(* Logix 5000 project; controller Receptivo vendor 1 type 14 code 106 rev 30.11; software revision 30.00; part 8 of 10 *)
(* tags used below, declared in another part *)
   Cantidad_de_Productos : DINT;
   codigo_capturado_1 : BOOL;
   codigo_capturado_2 : BOOL;
   codigo_capturado_3 : BOOL;
   codigo_capturado_4 : BOOL;
   Cont_Prod_1 : DINT;
   Cont_Prod_2 : DINT;
   Cont_Prod_3 : DINT;
   Cont_Prod_4 : DINT;
   Datos_1_Manual : BOOL;
   Datos_2_Manual : BOOL;
   Datos_3_Manual : BOOL;
   Datos_4_Manual : BOOL;
   EAN14_1 : Codigo_Barras;
   EAN14_2 : Codigo_Barras;
   EAN14_3 : Codigo_Barras;
   EAN14_4 : Codigo_Barras;
   Estacion_1_GCola_1 : UDT_COLA;
   Estacion_1_General : UDT_GENERAL;
   Estacion_2_GCola_1 : UDT_COLA;
   Estacion_2_General : UDT_GENERAL;
   Estacion_3_GCola_1 : UDT_COLA;
   Estacion_3_General : UDT_GENERAL;
   Estacion_4_GCola_1 : UDT_COLA;
   Estacion_4_General : UDT_GENERAL;
   No_existe : Descripcion;
   PB_Tare_Station_1 : BOOL;
   PB_Tare_Station_2 : BOOL;
   PESO_REAL_1 : DINT;
   PESO_REAL_2 : DINT;
   Producto1 : UDT_Inventario;
   Producto2 : UDT_Inventario;
   Producto3 : UDT_Inventario;
   Producto4 : UDT_Inventario;
   Producto_Codigo_Aceite_1 : DINT;
   Producto_Codigo_Aceite_2 : DINT;
   Producto_Codigo_Aceite_3 : DINT;
   Producto_Codigo_Aceite_4 : DINT;
   Productos : UDT_Maestro[300];
   QAD_1 : STRING;
   QAD_2 : STRING;
   QAD_3 : STRING;
   QAD_4 : STRING;
   Sin_Codigo : UDT_QAD;
   Station1_Tare_OK : BOOL;
   Station2_Tare_OK : BOOL;
   Tara_Fecha_Estacion_1 : Hora_y_Fecha;
   Tara_Fecha_Estacion_2 : Hora_y_Fecha;
   Tare_Station_1_Write : DINT;
   Tare_Station_2_Write : DINT;
   WPM1_Heartbeat : DINT;
   WPM1_Heartbeat_Error : BOOL;
   WPM1_Status : WPM_Status;
   WPM2_Heartbeat : DINT;
   WPM2_Heartbeat_Error : BOOL;
   WPM2_Status : WPM_Status;
   WPM_1_Selected : DINT;
   WPM_1_Status_Aux : DINT;
   WPM_2_COUNT_ANTERIOR : DINT;
   WPM_2_Selected : DINT;
   WPM_2_Status_Aux : DINT;
   Zero : DINT;

PROGRAM Manejo_Productos   (* main routine Inicial_Productos *)
VAR
   Final_captura_1 : BOOL;
   Final_captura_2 : BOOL;
   Final_captura_3 : BOOL;
   Final_captura_4 : BOOL;
   index_1 : DINT := 1;
   index_2 : DINT := 1;
   index_3 : DINT := 1;
   index_4 : DINT := 1;
   limite : BOOL := 1;
   ons_busca_1 : BOOL;
   ons_busca_2 : BOOL;
   ons_busca_3 : BOOL;
   ons_busca_4 : BOOL;
   ONS_CAPTURA : BOOL := 1;
   ONS_CAPTURA2 : BOOL;
   ONS_CAPTURA3 : BOOL;
   ONS_CAPTURA4 : BOOL;
   ons_captura_1 : BOOL;
   ons_dato_manual_1 : BOOL;
   ons_search : BOOL;
   vacio : STRING;
   victor : BOOL := 1;
END_VAR

ROUTINE Buscar_Productos_1   (* ladder *)
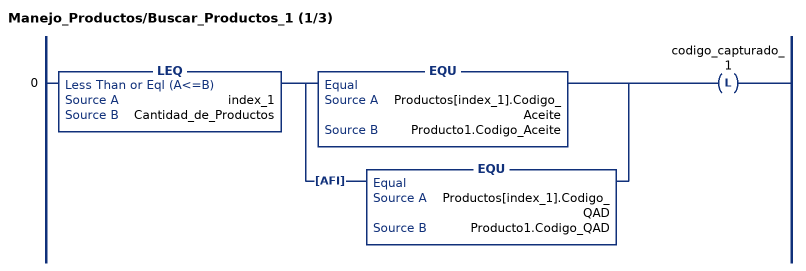
   0: LEQ(index_1,Cantidad_de_Productos)[EQU(Productos[index_1].Codigo_Aceite,Producto1.Codigo_Aceite) ,AFI() EQU(Productos[index_1].Codigo_QAD,Producto1.Codigo_QAD) ]OTL(codigo_capturado_1);
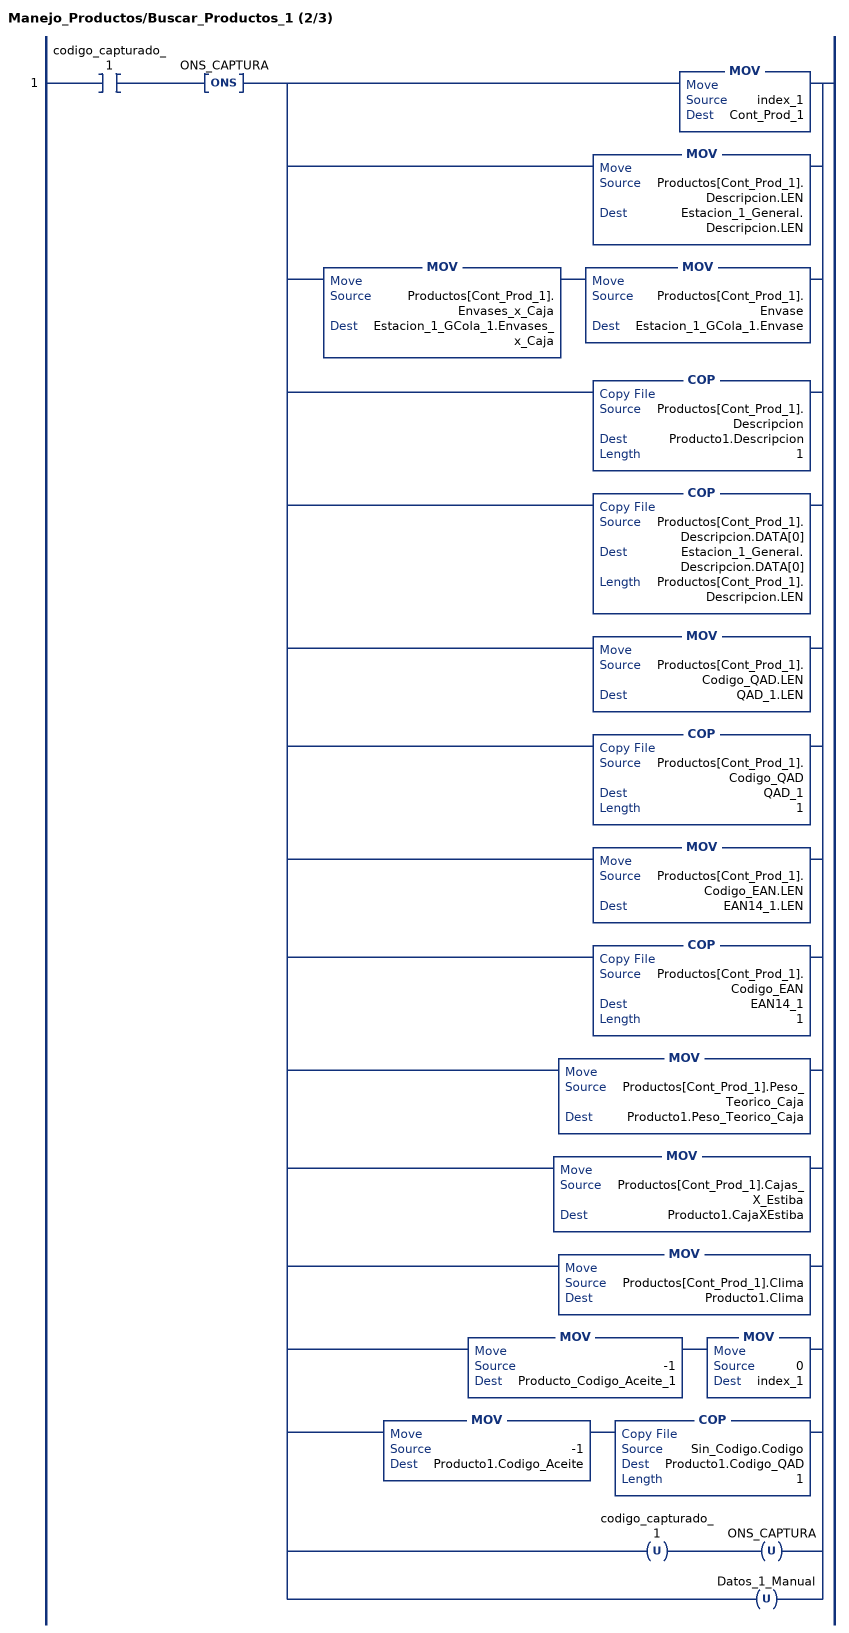
   1: XIC(codigo_capturado_1)ONS(ONS_CAPTURA)[MOV(index_1,Cont_Prod_1) ,MOV(Productos[Cont_Prod_1].Descripcion.LEN,Estacion_1_General.Descripcion.LEN) ,MOV(Productos[Cont_Prod_1].Envases_x_Caja,Estacion_1_GCola_1.Envases_x_Caja) MOV(Productos[Cont_Prod_1].Envase,Estacion_1_GCola_1.Envase) ,COP(Productos[Cont_Prod_1].Descripcion,Producto1.Descripcion,1) ,COP(Productos[Cont_Prod_1].Descripcion.DATA[0],Estacion_1_General.Descripcion.DATA[0],Productos[Cont_Prod_1].Descripcion.LEN) ,MOV(Productos[Cont_Prod_1].Codigo_QAD.LEN,QAD_1.LEN) ,COP(Productos[Cont_Prod_1].Codigo_QAD,QAD_1,1) ,MOV(Productos[Cont_Prod_1].Codigo_EAN.LEN,EAN14_1.LEN) ,COP(Productos[Cont_Prod_1].Codigo_EAN,EAN14_1,1) ,MOV(Productos[Cont_Prod_1].Peso_Teorico_Caja,Producto1.Peso_Teorico_Caja) ,MOV(Productos[Cont_Prod_1].Cajas_X_Estiba,Producto1.CajaXEstiba) ,MOV(Productos[Cont_Prod_1].Clima,Producto1.Clima) ,MOV(-1,Producto_Codigo_Aceite_1) MOV(0,index_1) ,MOV(-1,Producto1.Codigo_Aceite) COP(Sin_Codigo.Codigo,Producto1.Codigo_QAD,1) ,OTU(codigo_capturado_1) OTU(ONS_CAPTURA) ,OTU(Datos_1_Manual) ];
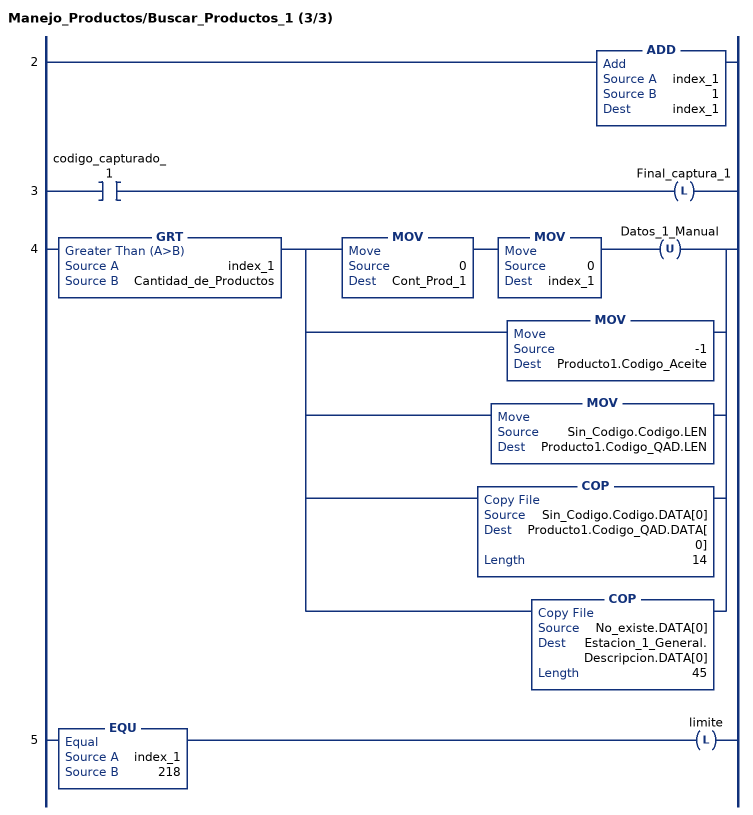
   2: ADD(index_1,1,index_1);
   3: XIC(codigo_capturado_1)OTL(Final_captura_1);
   4: GRT(index_1,Cantidad_de_Productos)[MOV(0,Cont_Prod_1) MOV(0,index_1) OTU(Datos_1_Manual) ,MOV(-1,Producto1.Codigo_Aceite) ,MOV(Sin_Codigo.Codigo.LEN,Producto1.Codigo_QAD.LEN) ,COP(Sin_Codigo.Codigo.DATA[0],Producto1.Codigo_QAD.DATA[0],14) ,COP(No_existe.DATA[0],Estacion_1_General.Descripcion.DATA[0],45) ];
   5: EQU(index_1,218)OTL(limite);
END_ROUTINE

ROUTINE Buscar_Productos_2   (* ladder *)
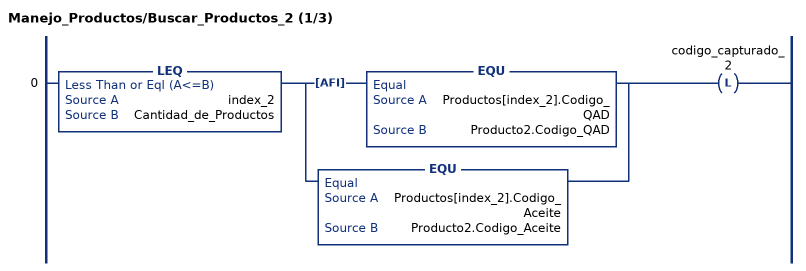
   0: LEQ(index_2,Cantidad_de_Productos)[AFI() EQU(Productos[index_2].Codigo_QAD,Producto2.Codigo_QAD) ,EQU(Productos[index_2].Codigo_Aceite,Producto2.Codigo_Aceite) ]OTL(codigo_capturado_2);
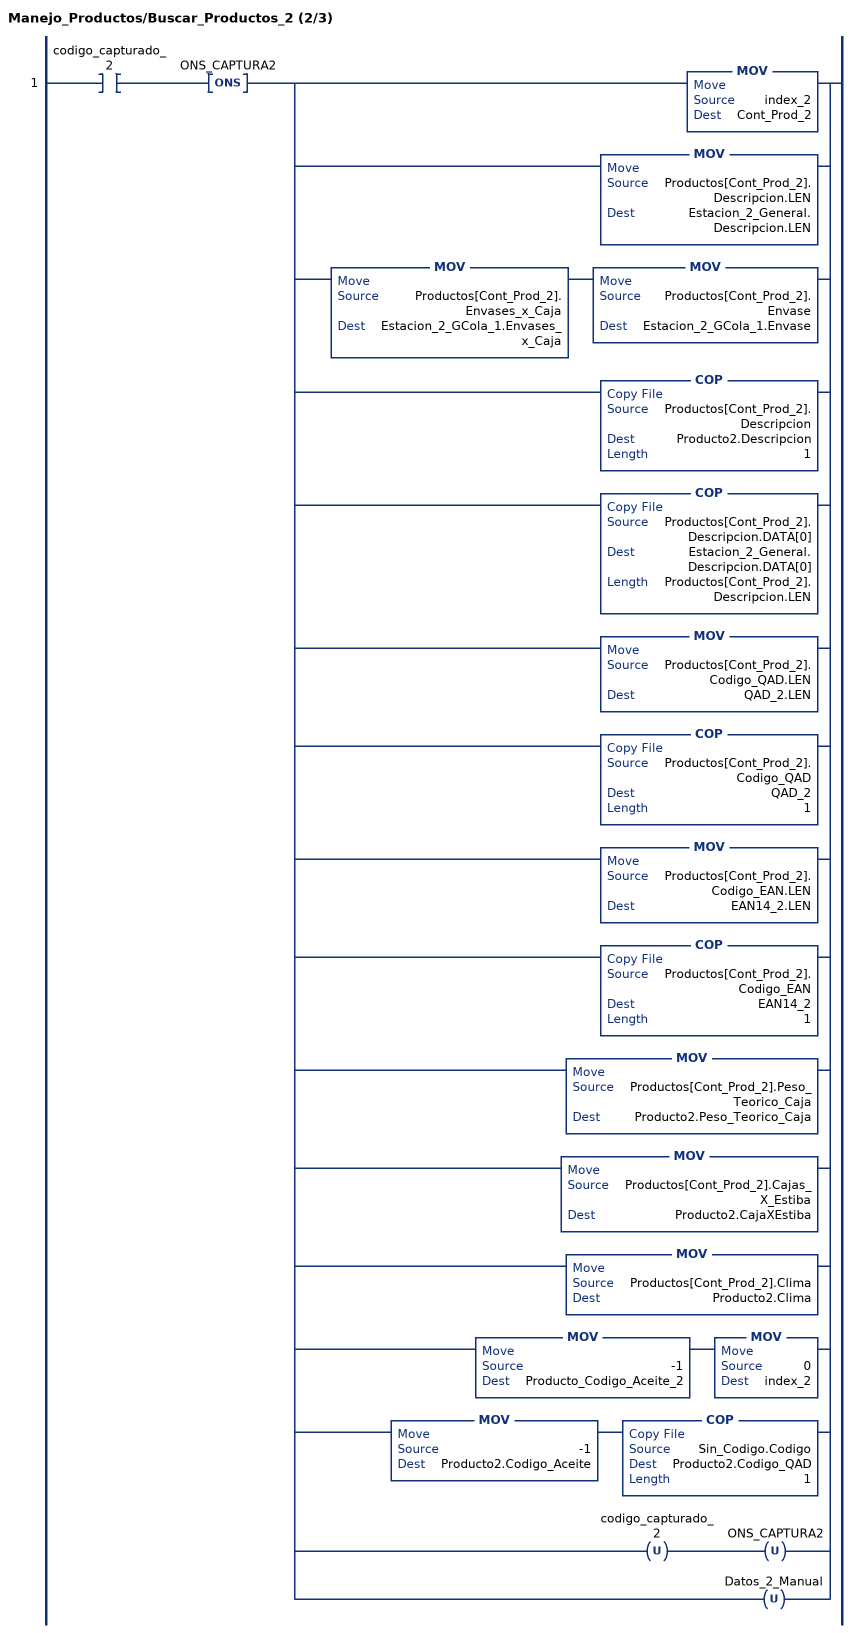
   1: XIC(codigo_capturado_2)ONS(ONS_CAPTURA2)[MOV(index_2,Cont_Prod_2) ,MOV(Productos[Cont_Prod_2].Descripcion.LEN,Estacion_2_General.Descripcion.LEN) ,MOV(Productos[Cont_Prod_2].Envases_x_Caja,Estacion_2_GCola_1.Envases_x_Caja) MOV(Productos[Cont_Prod_2].Envase,Estacion_2_GCola_1.Envase) ,COP(Productos[Cont_Prod_2].Descripcion,Producto2.Descripcion,1) ,COP(Productos[Cont_Prod_2].Descripcion.DATA[0],Estacion_2_General.Descripcion.DATA[0],Productos[Cont_Prod_2].Descripcion.LEN) ,MOV(Productos[Cont_Prod_2].Codigo_QAD.LEN,QAD_2.LEN) ,COP(Productos[Cont_Prod_2].Codigo_QAD,QAD_2,1) ,MOV(Productos[Cont_Prod_2].Codigo_EAN.LEN,EAN14_2.LEN) ,COP(Productos[Cont_Prod_2].Codigo_EAN,EAN14_2,1) ,MOV(Productos[Cont_Prod_2].Peso_Teorico_Caja,Producto2.Peso_Teorico_Caja) ,MOV(Productos[Cont_Prod_2].Cajas_X_Estiba,Producto2.CajaXEstiba) ,MOV(Productos[Cont_Prod_2].Clima,Producto2.Clima) ,MOV(-1,Producto_Codigo_Aceite_2) MOV(0,index_2) ,MOV(-1,Producto2.Codigo_Aceite) COP(Sin_Codigo.Codigo,Producto2.Codigo_QAD,1) ,OTU(codigo_capturado_2) OTU(ONS_CAPTURA2) ,OTU(Datos_2_Manual) ];
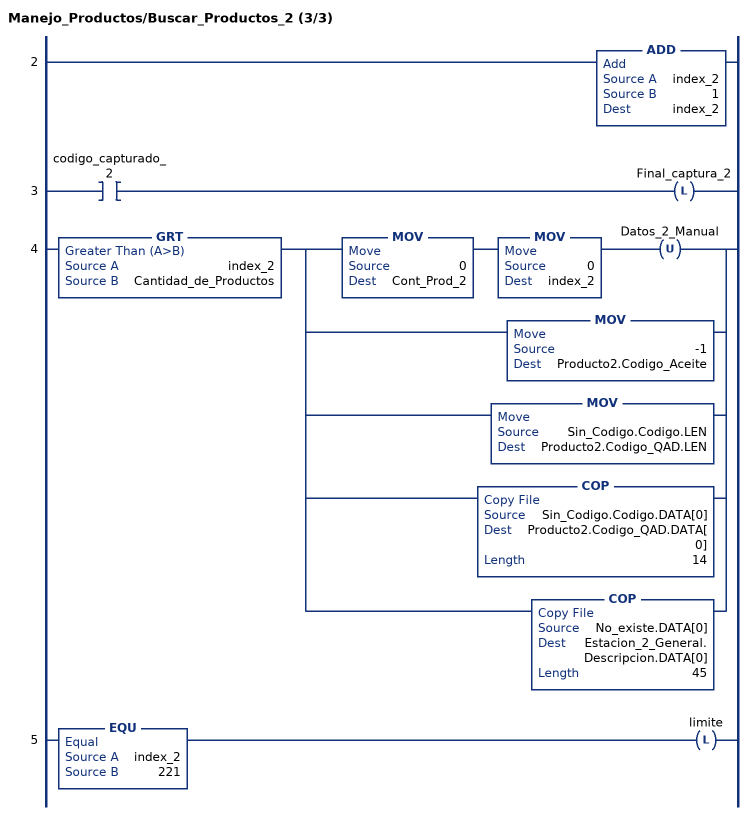
   2: ADD(index_2,1,index_2);
   3: XIC(codigo_capturado_2)OTL(Final_captura_2);
   4: GRT(index_2,Cantidad_de_Productos)[MOV(0,Cont_Prod_2) MOV(0,index_2) OTU(Datos_2_Manual) ,MOV(-1,Producto2.Codigo_Aceite) ,MOV(Sin_Codigo.Codigo.LEN,Producto2.Codigo_QAD.LEN) ,COP(Sin_Codigo.Codigo.DATA[0],Producto2.Codigo_QAD.DATA[0],14) ,COP(No_existe.DATA[0],Estacion_2_General.Descripcion.DATA[0],45) ];
   5: EQU(index_2,221)OTL(limite);
END_ROUTINE

ROUTINE Buscar_Productos_3   (* ladder *)
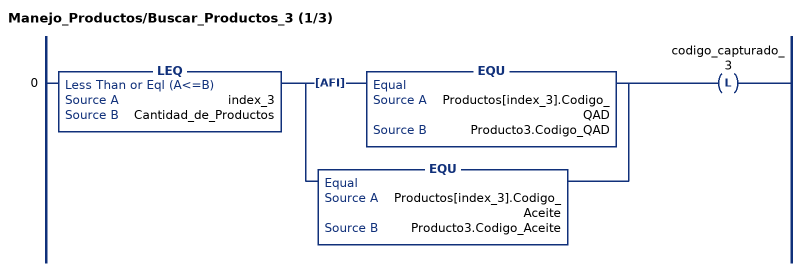
   0: LEQ(index_3,Cantidad_de_Productos)[AFI() EQU(Productos[index_3].Codigo_QAD,Producto3.Codigo_QAD) ,EQU(Productos[index_3].Codigo_Aceite,Producto3.Codigo_Aceite) ]OTL(codigo_capturado_3);
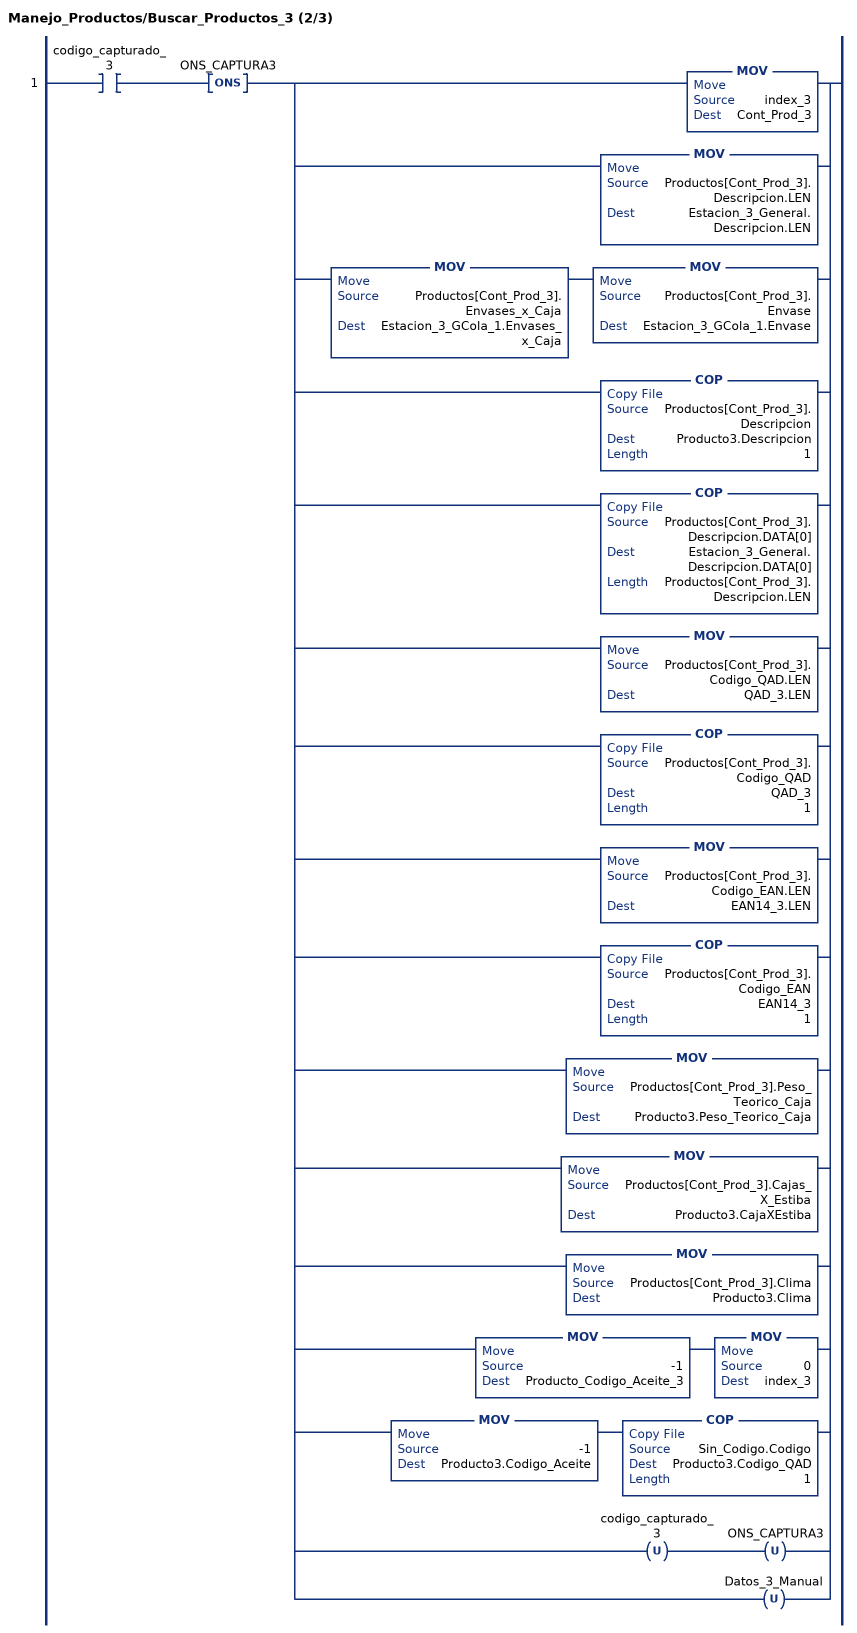
   1: XIC(codigo_capturado_3)ONS(ONS_CAPTURA3)[MOV(index_3,Cont_Prod_3) ,MOV(Productos[Cont_Prod_3].Descripcion.LEN,Estacion_3_General.Descripcion.LEN) ,MOV(Productos[Cont_Prod_3].Envases_x_Caja,Estacion_3_GCola_1.Envases_x_Caja) MOV(Productos[Cont_Prod_3].Envase,Estacion_3_GCola_1.Envase) ,COP(Productos[Cont_Prod_3].Descripcion,Producto3.Descripcion,1) ,COP(Productos[Cont_Prod_3].Descripcion.DATA[0],Estacion_3_General.Descripcion.DATA[0],Productos[Cont_Prod_3].Descripcion.LEN) ,MOV(Productos[Cont_Prod_3].Codigo_QAD.LEN,QAD_3.LEN) ,COP(Productos[Cont_Prod_3].Codigo_QAD,QAD_3,1) ,MOV(Productos[Cont_Prod_3].Codigo_EAN.LEN,EAN14_3.LEN) ,COP(Productos[Cont_Prod_3].Codigo_EAN,EAN14_3,1) ,MOV(Productos[Cont_Prod_3].Peso_Teorico_Caja,Producto3.Peso_Teorico_Caja) ,MOV(Productos[Cont_Prod_3].Cajas_X_Estiba,Producto3.CajaXEstiba) ,MOV(Productos[Cont_Prod_3].Clima,Producto3.Clima) ,MOV(-1,Producto_Codigo_Aceite_3) MOV(0,index_3) ,MOV(-1,Producto3.Codigo_Aceite) COP(Sin_Codigo.Codigo,Producto3.Codigo_QAD,1) ,OTU(codigo_capturado_3) OTU(ONS_CAPTURA3) ,OTU(Datos_3_Manual) ];
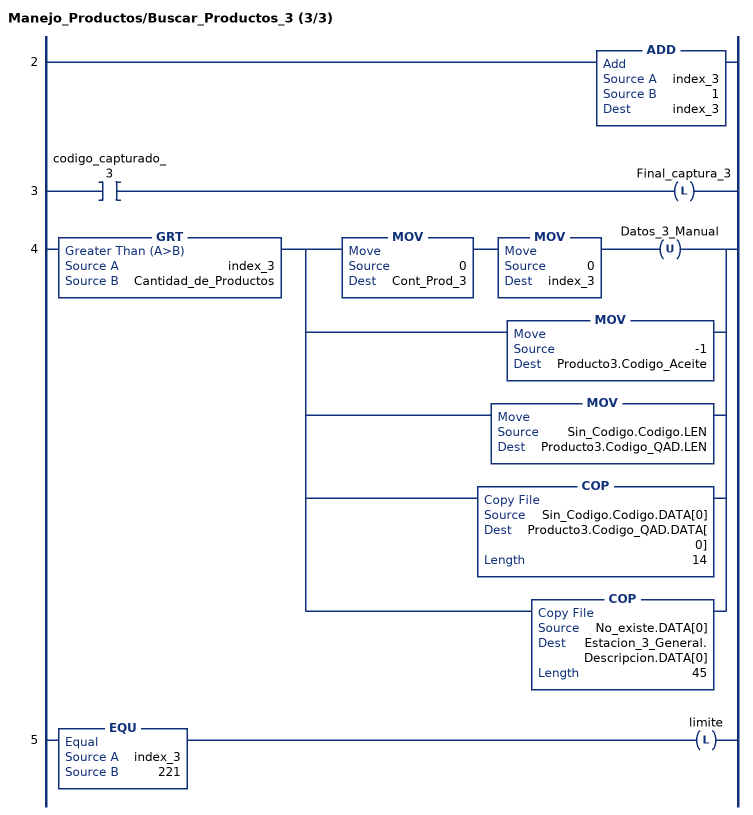
   2: ADD(index_3,1,index_3);
   3: XIC(codigo_capturado_3)OTL(Final_captura_3);
   4: GRT(index_3,Cantidad_de_Productos)[MOV(0,Cont_Prod_3) MOV(0,index_3) OTU(Datos_3_Manual) ,MOV(-1,Producto3.Codigo_Aceite) ,MOV(Sin_Codigo.Codigo.LEN,Producto3.Codigo_QAD.LEN) ,COP(Sin_Codigo.Codigo.DATA[0],Producto3.Codigo_QAD.DATA[0],14) ,COP(No_existe.DATA[0],Estacion_3_General.Descripcion.DATA[0],45) ];
   5: EQU(index_3,221)OTL(limite);
END_ROUTINE

ROUTINE Buscar_Productos_4   (* ladder *)
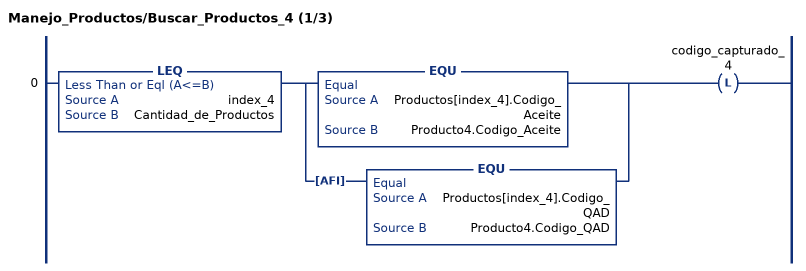
   0: LEQ(index_4,Cantidad_de_Productos)[EQU(Productos[index_4].Codigo_Aceite,Producto4.Codigo_Aceite) ,AFI() EQU(Productos[index_4].Codigo_QAD,Producto4.Codigo_QAD) ]OTL(codigo_capturado_4);
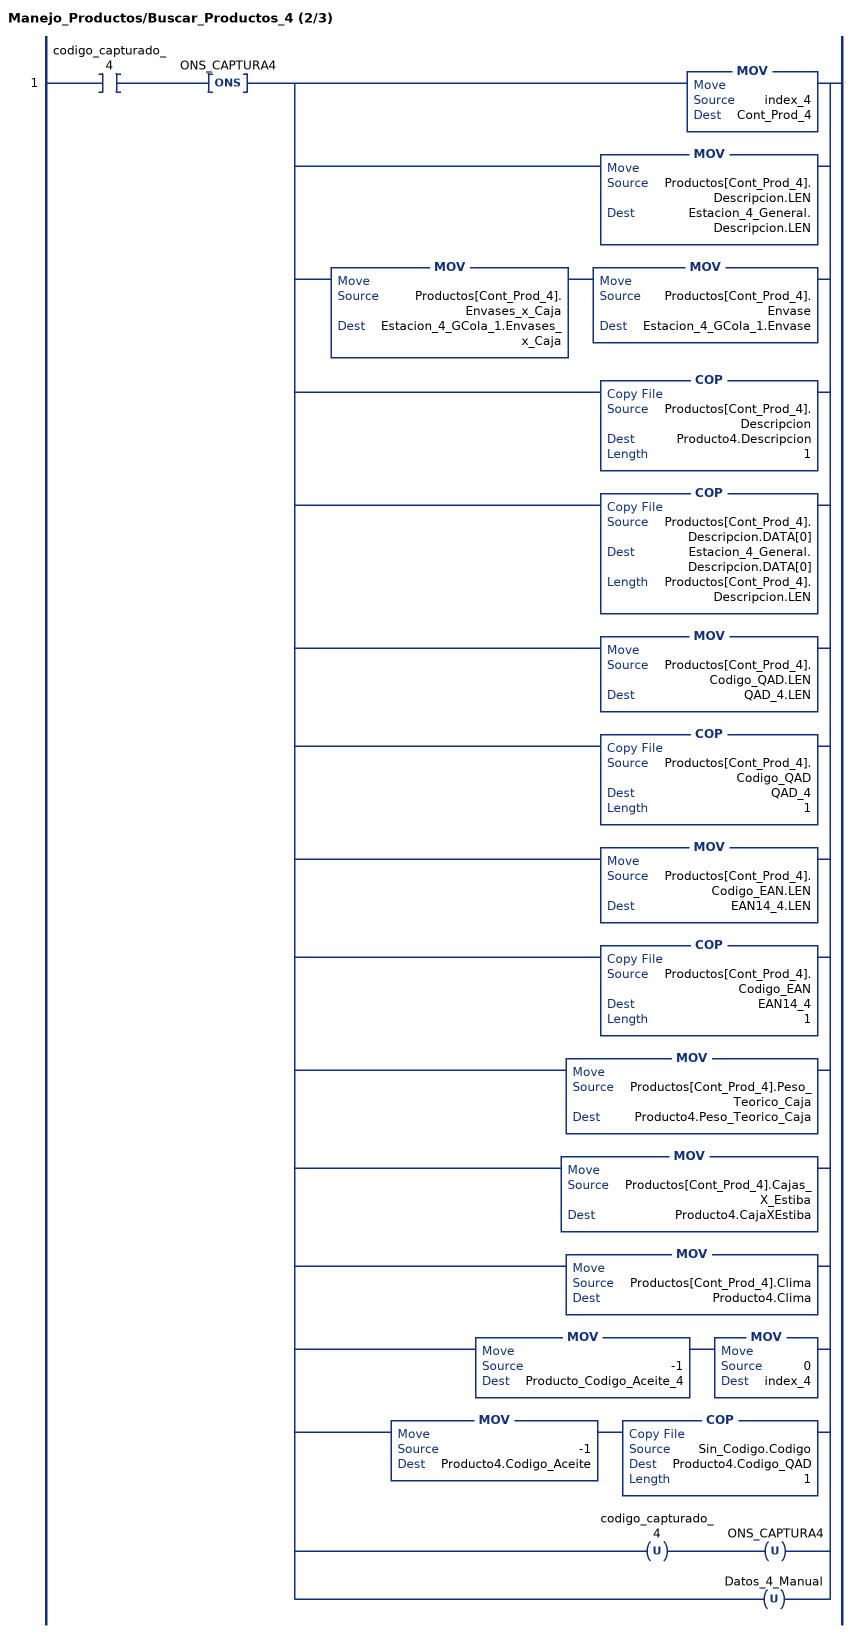
   1: XIC(codigo_capturado_4)ONS(ONS_CAPTURA4)[MOV(index_4,Cont_Prod_4) ,MOV(Productos[Cont_Prod_4].Descripcion.LEN,Estacion_4_General.Descripcion.LEN) ,MOV(Productos[Cont_Prod_4].Envases_x_Caja,Estacion_4_GCola_1.Envases_x_Caja) MOV(Productos[Cont_Prod_4].Envase,Estacion_4_GCola_1.Envase) ,COP(Productos[Cont_Prod_4].Descripcion,Producto4.Descripcion,1) ,COP(Productos[Cont_Prod_4].Descripcion.DATA[0],Estacion_4_General.Descripcion.DATA[0],Productos[Cont_Prod_4].Descripcion.LEN) ,MOV(Productos[Cont_Prod_4].Codigo_QAD.LEN,QAD_4.LEN) ,COP(Productos[Cont_Prod_4].Codigo_QAD,QAD_4,1) ,MOV(Productos[Cont_Prod_4].Codigo_EAN.LEN,EAN14_4.LEN) ,COP(Productos[Cont_Prod_4].Codigo_EAN,EAN14_4,1) ,MOV(Productos[Cont_Prod_4].Peso_Teorico_Caja,Producto4.Peso_Teorico_Caja) ,MOV(Productos[Cont_Prod_4].Cajas_X_Estiba,Producto4.CajaXEstiba) ,MOV(Productos[Cont_Prod_4].Clima,Producto4.Clima) ,MOV(-1,Producto_Codigo_Aceite_4) MOV(0,index_4) ,MOV(-1,Producto4.Codigo_Aceite) COP(Sin_Codigo.Codigo,Producto4.Codigo_QAD,1) ,OTU(codigo_capturado_4) OTU(ONS_CAPTURA4) ,OTU(Datos_4_Manual) ];
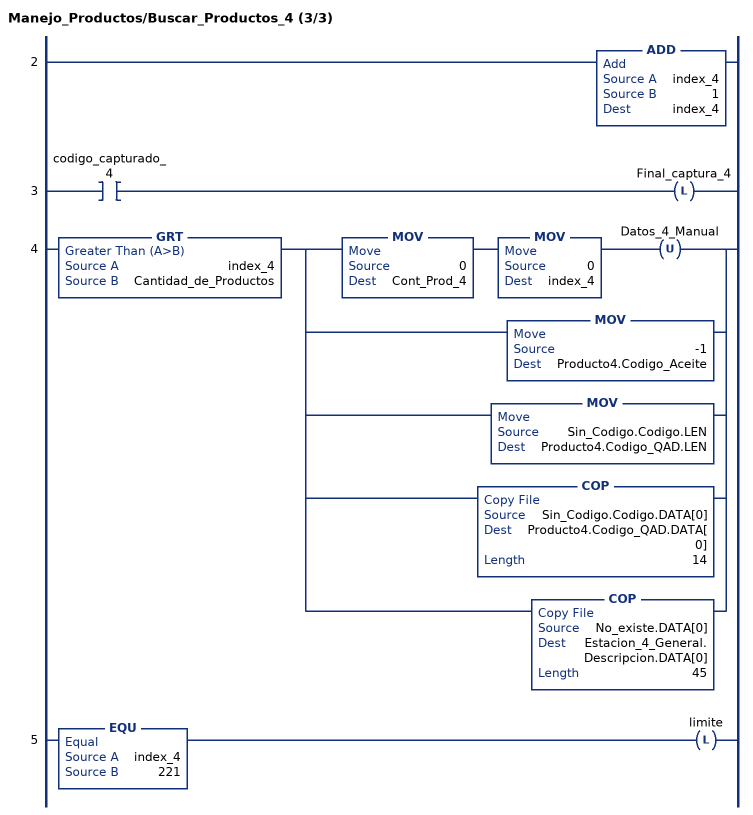
   2: ADD(index_4,1,index_4);
   3: XIC(codigo_capturado_4)OTL(Final_captura_4);
   4: GRT(index_4,Cantidad_de_Productos)[MOV(0,Cont_Prod_4) MOV(0,index_4) OTU(Datos_4_Manual) ,MOV(-1,Producto4.Codigo_Aceite) ,MOV(Sin_Codigo.Codigo.LEN,Producto4.Codigo_QAD.LEN) ,COP(Sin_Codigo.Codigo.DATA[0],Producto4.Codigo_QAD.DATA[0],14) ,COP(No_existe.DATA[0],Estacion_4_General.Descripcion.DATA[0],45) ];
   5: EQU(index_4,221)OTL(limite);
END_ROUTINE

ROUTINE Inicial_Productos   (* ladder *)
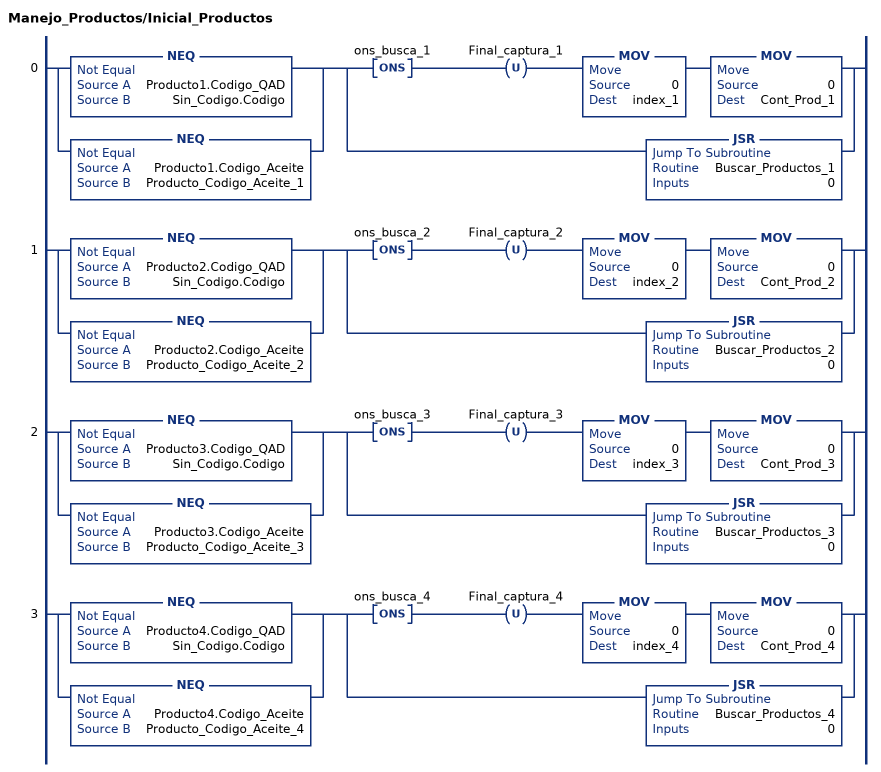
   0: [NEQ(Producto1.Codigo_QAD,Sin_Codigo.Codigo) ,NEQ(Producto1.Codigo_Aceite,Producto_Codigo_Aceite_1) ][ONS(ons_busca_1) OTU(Final_captura_1) MOV(0,index_1) MOV(0,Cont_Prod_1) ,JSR(Buscar_Productos_1,0) ];
   1: [NEQ(Producto2.Codigo_QAD,Sin_Codigo.Codigo) ,NEQ(Producto2.Codigo_Aceite,Producto_Codigo_Aceite_2) ][ONS(ons_busca_2) OTU(Final_captura_2) MOV(0,index_2) MOV(0,Cont_Prod_2) ,JSR(Buscar_Productos_2,0) ];
   2: [NEQ(Producto3.Codigo_QAD,Sin_Codigo.Codigo) ,NEQ(Producto3.Codigo_Aceite,Producto_Codigo_Aceite_3) ][ONS(ons_busca_3) OTU(Final_captura_3) MOV(0,index_3) MOV(0,Cont_Prod_3) ,JSR(Buscar_Productos_3,0) ];
   3: [NEQ(Producto4.Codigo_QAD,Sin_Codigo.Codigo) ,NEQ(Producto4.Codigo_Aceite,Producto_Codigo_Aceite_4) ][ONS(ons_busca_4) OTU(Final_captura_4) MOV(0,index_4) MOV(0,Cont_Prod_4) ,JSR(Buscar_Productos_4,0) ];
END_ROUTINE
END_PROGRAM

PROGRAM Pesaje   (* main routine Pesaje_Principal *)
VAR
   Command_Status : DINT := 32768;
   Conteo_Gway_Anterior : DINT;
   Gway_Error : BOOL := 1;
   GWay_Heartbeat : DINT := 3;
   Gway_Status : DINT;
   ons_conteo_gway : BOOL;
   ons_gway_change : BOOL := 1;
   ons_nuevo_dia : BOOL;
   ons_pesaje_1 : BOOL;
   ons_tare_station_1 : BOOL;
   ons_tare_station_2 : BOOL;
   ons_tare_station_3 : BOOL;
   ons_wpm1 : BOOL;
   ons_wpm2 : BOOL;
   ons_wpm3 : BOOL;
   ons_wpm4 : BOOL;
   Timer_Gway_1 : TIMER := (PRE := 1000);
   Timer_Gway_2 : TIMER := (PRE := 1000);
   Timer_Gway_3 : TIMER := (PRE := 1000);
   Timer_Gway_4 : TIMER := (PRE := 1000, ACC := 11, EN := 1, TT := 1);
   Timer_Gway_Hearbeat : TIMER[4] := ([0].PRE := 3000, [1].PRE := 3000, [2].PRE := 3000, [3].PRE := 3000, [3].ACC := 87, [3].EN := 1, [3].TT := 1);
   Timer_Tare_Station_1 : TIMER := (PRE := 3000);
   Timer_Tare_Station_1_aux : BOOL;
   Timer_Tare_Station_2 : TIMER := (PRE := 3000);
   Timer_Tare_Station_2_aux : BOOL;
   Timer_Tare_Station_3 : TIMER := (PRE := 3000);
   Timer_Tare_Station_3_aux : BOOL;
   Timer_Tare_Station_4 : TIMER := (PRE := 3000);
   Timer_Tare_Station_4_aux : BOOL;
   Timer_WPM1_Heartbeat : TIMER[8] := ([0].PRE := 3000, [1].PRE := 3000, [2].PRE := 3000, [3].PRE := 3000, [4].PRE := 3000, [4].ACC := 93, [4].EN := 1, [4].TT := 1, [5].PRE := 3000, [6].PRE := 3000, [7].PRE := 3000);
   Timer_WPM2_Heartbeat : TIMER[8] := ([0].PRE := 3000, [1].PRE := 3000, [1].ACC := 5, [1].EN := 1, [1].TT := 1, [2].PRE := 3000, [3].PRE := 3000, [4].PRE := 3000, [5].PRE := 3000, [6].PRE := 3000, [7].PRE := 3000);
   Timer_WPM3_Heartbeat : TIMER[8] := ([0].PRE := 3000, [1].PRE := 3000, [2].PRE := 3000, [3].PRE := 3000, [4].PRE := 3000, [5].PRE := 3000, [6].PRE := 3000, [7].PRE := 3000, [7].ACC := 75, [7].EN := 1, [7].TT := 1);
   Timer_WPM4_Heartbeat : TIMER[8] := ([0].PRE := 3000, [1].PRE := 3000, [2].PRE := 3000, [3].PRE := 3000, [4].PRE := 3000, [5].PRE := 3000, [6].PRE := 3000, [6].ACC := 82, [6].EN := 1, [6].TT := 1, [7].PRE := 3000);
   WPM2_No_Count : BOOL := 1;
   WPM_1_COUNT_ANTERIOR : DINT := 4;
   WPM_3_COUNT_ANTERIOR : DINT := 7;
   WPM_4_COUNT_ANTERIOR : DINT := 6;
END_VAR

ROUTINE Control_Pesaje_1   (* ladder *)
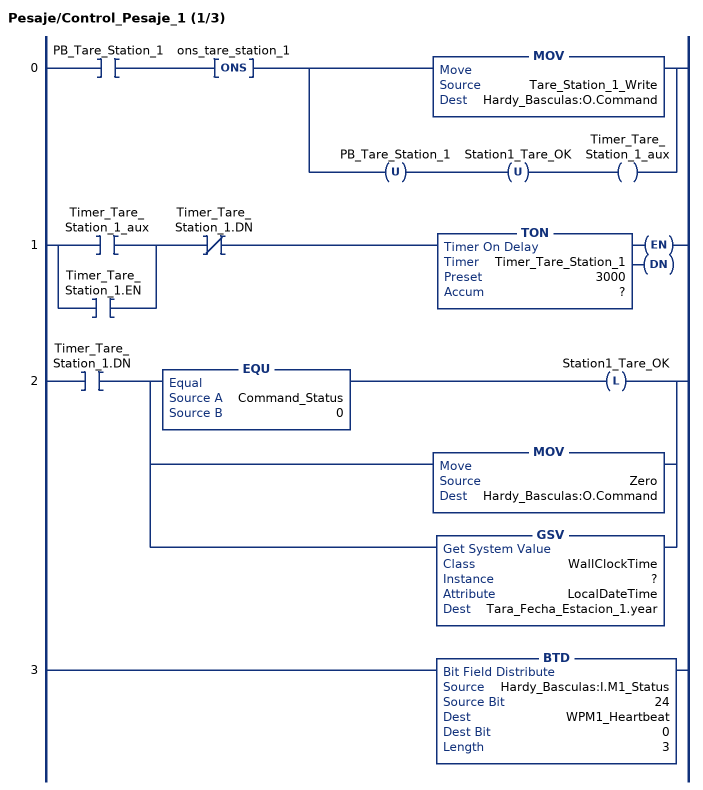
   0: XIC(PB_Tare_Station_1)ONS(ons_tare_station_1)[MOV(Tare_Station_1_Write,Hardy_Basculas:O.Command) ,OTU(PB_Tare_Station_1) OTU(Station1_Tare_OK) OTE(Timer_Tare_Station_1_aux) ];
   1: [XIC(Timer_Tare_Station_1_aux) ,XIC(Timer_Tare_Station_1.EN) ]XIO(Timer_Tare_Station_1.DN)TON(Timer_Tare_Station_1,?,?);
   2: XIC(Timer_Tare_Station_1.DN)[EQU(Command_Status,0) OTL(Station1_Tare_OK) ,MOV(Zero,Hardy_Basculas:O.Command) ,GSV(WallClockTime,?,LocalDateTime,Tara_Fecha_Estacion_1.year) ];
   3: BTD(Hardy_Basculas:I.M1_Status,24,WPM1_Heartbeat,0,3);
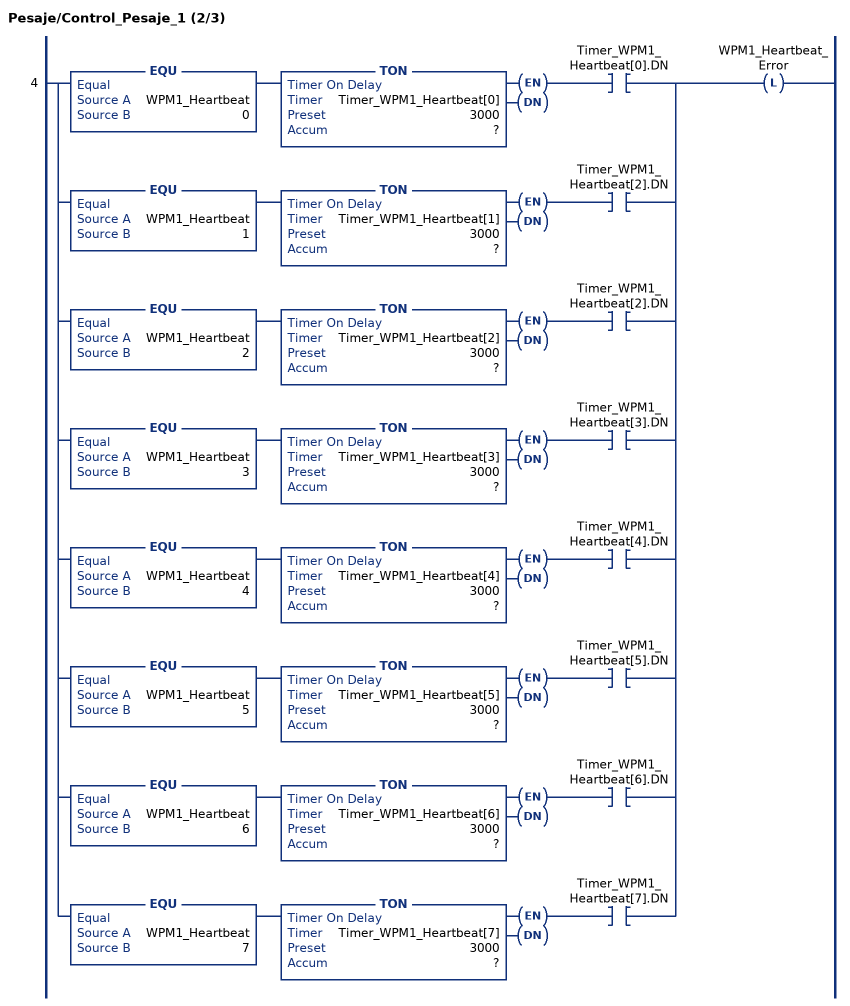
   4: [EQU(WPM1_Heartbeat,0) TON(Timer_WPM1_Heartbeat[0],?,?) XIC(Timer_WPM1_Heartbeat[0].DN) ,EQU(WPM1_Heartbeat,1) TON(Timer_WPM1_Heartbeat[1],?,?) XIC(Timer_WPM1_Heartbeat[2].DN) ,EQU(WPM1_Heartbeat,2) TON(Timer_WPM1_Heartbeat[2],?,?) XIC(Timer_WPM1_Heartbeat[2].DN) ,EQU(WPM1_Heartbeat,3) TON(Timer_WPM1_Heartbeat[3],?,?) XIC(Timer_WPM1_Heartbeat[3].DN) ,EQU(WPM1_Heartbeat,4) TON(Timer_WPM1_Heartbeat[4],?,?) XIC(Timer_WPM1_Heartbeat[4].DN) ,EQU(WPM1_Heartbeat,5) TON(Timer_WPM1_Heartbeat[5],?,?) XIC(Timer_WPM1_Heartbeat[5].DN) ,EQU(WPM1_Heartbeat,6) TON(Timer_WPM1_Heartbeat[6],?,?) XIC(Timer_WPM1_Heartbeat[6].DN) ,EQU(WPM1_Heartbeat,7) TON(Timer_WPM1_Heartbeat[7],?,?) XIC(Timer_WPM1_Heartbeat[7].DN) ]OTL(WPM1_Heartbeat_Error);
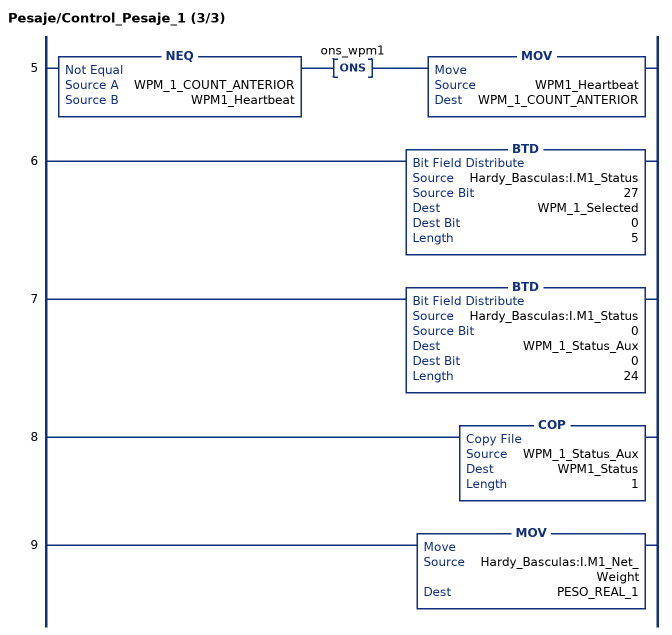
   5: NEQ(WPM_1_COUNT_ANTERIOR,WPM1_Heartbeat)ONS(ons_wpm1)MOV(WPM1_Heartbeat,WPM_1_COUNT_ANTERIOR);
   6: BTD(Hardy_Basculas:I.M1_Status,27,WPM_1_Selected,0,5);
   7: BTD(Hardy_Basculas:I.M1_Status,0,WPM_1_Status_Aux,0,24);
   8: COP(WPM_1_Status_Aux,WPM1_Status,1);
   9: MOV(Hardy_Basculas:I.M1_Net_Weight,PESO_REAL_1);
END_ROUTINE

ROUTINE Control_Pesaje_2   (* ladder *)
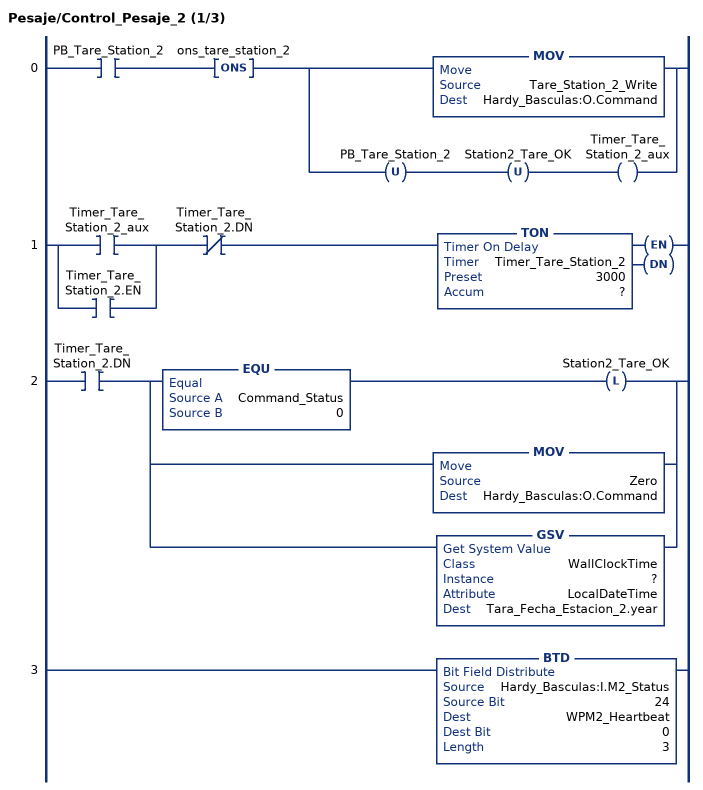
   0: XIC(PB_Tare_Station_2)ONS(ons_tare_station_2)[MOV(Tare_Station_2_Write,Hardy_Basculas:O.Command) ,OTU(PB_Tare_Station_2) OTU(Station2_Tare_OK) OTE(Timer_Tare_Station_2_aux) ];
   1: [XIC(Timer_Tare_Station_2_aux) ,XIC(Timer_Tare_Station_2.EN) ]XIO(Timer_Tare_Station_2.DN)TON(Timer_Tare_Station_2,?,?);
   2: XIC(Timer_Tare_Station_2.DN)[EQU(Command_Status,0) OTL(Station2_Tare_OK) ,MOV(Zero,Hardy_Basculas:O.Command) ,GSV(WallClockTime,?,LocalDateTime,Tara_Fecha_Estacion_2.year) ];
   3: BTD(Hardy_Basculas:I.M2_Status,24,WPM2_Heartbeat,0,3);
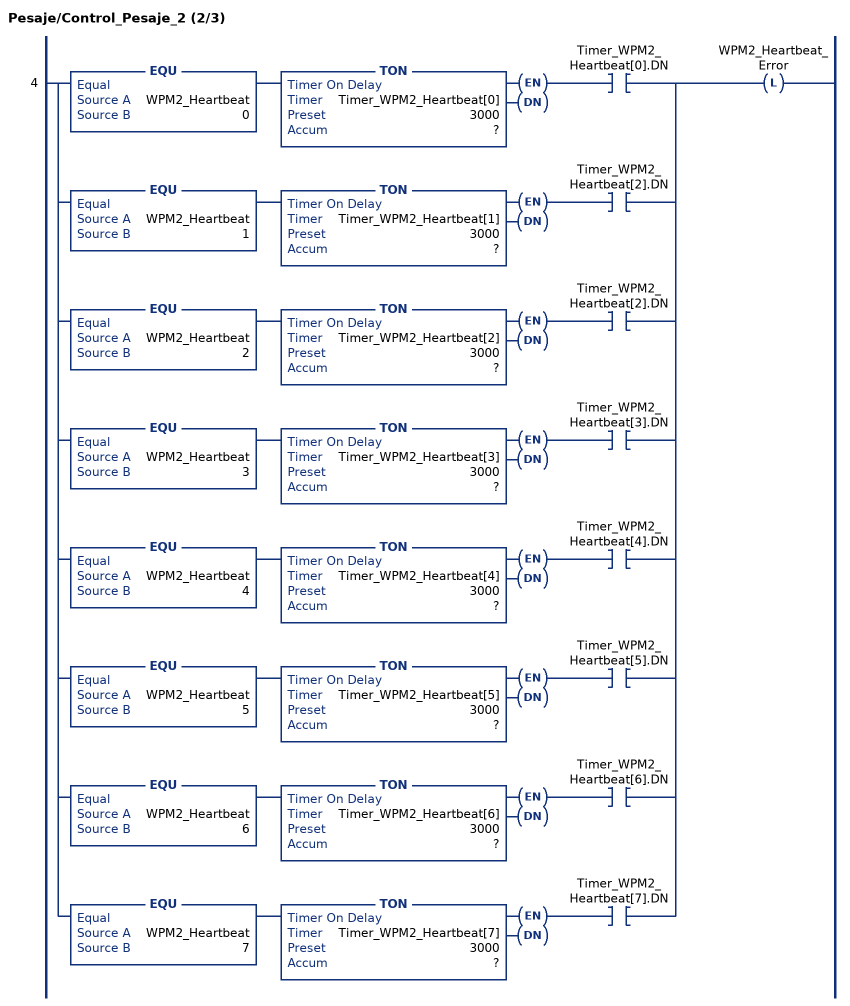
   4: [EQU(WPM2_Heartbeat,0) TON(Timer_WPM2_Heartbeat[0],?,?) XIC(Timer_WPM2_Heartbeat[0].DN) ,EQU(WPM2_Heartbeat,1) TON(Timer_WPM2_Heartbeat[1],?,?) XIC(Timer_WPM2_Heartbeat[2].DN) ,EQU(WPM2_Heartbeat,2) TON(Timer_WPM2_Heartbeat[2],?,?) XIC(Timer_WPM2_Heartbeat[2].DN) ,EQU(WPM2_Heartbeat,3) TON(Timer_WPM2_Heartbeat[3],?,?) XIC(Timer_WPM2_Heartbeat[3].DN) ,EQU(WPM2_Heartbeat,4) TON(Timer_WPM2_Heartbeat[4],?,?) XIC(Timer_WPM2_Heartbeat[4].DN) ,EQU(WPM2_Heartbeat,5) TON(Timer_WPM2_Heartbeat[5],?,?) XIC(Timer_WPM2_Heartbeat[5].DN) ,EQU(WPM2_Heartbeat,6) TON(Timer_WPM2_Heartbeat[6],?,?) XIC(Timer_WPM2_Heartbeat[6].DN) ,EQU(WPM2_Heartbeat,7) TON(Timer_WPM2_Heartbeat[7],?,?) XIC(Timer_WPM2_Heartbeat[7].DN) ]OTL(WPM2_Heartbeat_Error);
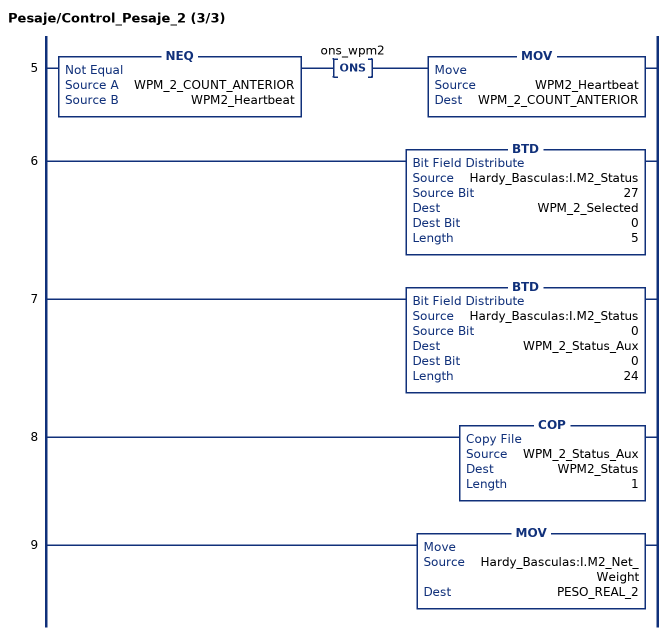
   5: NEQ(WPM_2_COUNT_ANTERIOR,WPM2_Heartbeat)ONS(ons_wpm2)MOV(WPM2_Heartbeat,WPM_2_COUNT_ANTERIOR);
   6: BTD(Hardy_Basculas:I.M2_Status,27,WPM_2_Selected,0,5);
   7: BTD(Hardy_Basculas:I.M2_Status,0,WPM_2_Status_Aux,0,24);
   8: COP(WPM_2_Status_Aux,WPM2_Status,1);
   9: MOV(Hardy_Basculas:I.M2_Net_Weight,PESO_REAL_2);
END_ROUTINE
